TYPE EtcMasterBase_62654B43 :
STRUCT
END_STRUCT
END_TYPE

(* stored: Version 1.2.0.0, ProductVersion 3.1.4024.11
   DUT EtcMasterBase_62654B43: Id {7e98699e-4ecf-4dbe-bd3d-8ef962272910} *)
